(* IEC 61131-3 sources: Word/plc-course/05-boolean-logic-and-fbd/labs/starter, 3 files *)

(* ---- 05-1-pump-permissive.st ---- *)
(* Lab 05-1: Transfer pump P-101 start permissive.
   Module 05 (Boolean logic and FBD). STARTER - the declarations are done for you;
   write the logic where it says TODO, then run:
     python3 tools/plctest.py 05-boolean-logic-and-fbd/labs/starter/05-1-pump-permissive.st

   The whole lab is combinational: no seal-in, latch or timer is needed. *)

PROGRAM TransferPump
  VAR (* I/O - addresses follow the OpenPLC convention *)
    SuctionOpenLS AT %IX0.0 : BOOL;  (* Suction valve XV-100 open limit switch (ZSO-100): TRUE = fully open *)
    LSL101_NC     AT %IX0.1 : BOOL;  (* Tank low-level switch LSL-101, NC: TRUE = level above the switch (healthy) *)
    MotorFault    AT %IX0.2 : BOOL;  (* Motor protection relay fault contact, NO: TRUE = protection tripped *)
    ManualSel     AT %IX0.3 : BOOL;  (* MAN-OFF-AUTO selector, MAN contact *)
    AutoSel       AT %IX0.4 : BOOL;  (* MAN-OFF-AUTO selector, AUTO contact *)
    Demand        AT %IX0.5 : BOOL;  (* Auto demand from the process: TRUE = liquid wanted *)
    ManualRunCmd  AT %IX0.6 : BOOL;  (* Manual run command, maintained: TRUE = run *)
    Pump          AT %QX0.0 : BOOL;  (* P-101 motor starter: TRUE = run *)
    PermissiveOK  AT %QX0.1 : BOOL;  (* White "Ready" lamp: all start permissives healthy *)
    SelectorFault AT %QX0.2 : BOOL;  (* Both selector contacts made at once *)
  END_VAR
  (* You may add your own internal variables in a separate VAR block here. *)

  (* TODO: replace these placeholder lines with your logic.
     (MATIEC needs at least one statement in a program body.) *)
  PermissiveOK := FALSE;
  SelectorFault := FALSE;
  Pump := FALSE;
END_PROGRAM

CONFIGURATION Config0
  RESOURCE Res0 ON PLC
    TASK MainTask(INTERVAL := T#10ms, PRIORITY := 0);
    PROGRAM Inst0 WITH MainTask : TransferPump;
  END_RESOURCE
END_CONFIGURATION

(* ---- 05-2-two-out-of-three-vote.st ---- *)
(* Lab 05-2: Two-out-of-three (2oo3) high-pressure trip vote.
   Module 05 (Boolean logic and FBD). STARTER - the declarations are done for you;
   write the logic where it says TODO, then run:
     python3 tools/plctest.py 05-boolean-logic-and-fbd/labs/starter/05-2-two-out-of-three-vote.st

   TRAINING EXERCISE ONLY - not a design for a real safety function. *)

PROGRAM TripVote
  VAR (* I/O - addresses follow the OpenPLC convention *)
    PSHH_A_NC   AT %IX0.0 : BOOL;  (* PSHH-101A, NC: TRUE = pressure below trip setting (healthy) *)
    PSHH_B_NC   AT %IX0.1 : BOOL;  (* PSHH-101B, NC: as above *)
    PSHH_C_NC   AT %IX0.2 : BOOL;  (* PSHH-101C, NC: as above *)
    Trip        AT %QX0.0 : BOOL;  (* TRUE = at least two channels demand a trip *)
    SDVSolenoid AT %QX0.1 : BOOL;  (* SDV-100 solenoid: TRUE = energised, valve held open *)
    Discrepancy AT %QX0.2 : BOOL;  (* TRUE = the three channels do not all agree *)
    DiscA       AT %QX0.3 : BOOL;  (* TRUE = channel A disagrees with B and C *)
    DiscB       AT %QX0.4 : BOOL;  (* TRUE = channel B disagrees with A and C *)
    DiscC       AT %QX0.5 : BOOL;  (* TRUE = channel C disagrees with A and B *)
  END_VAR
  (* You may add your own internal variables in a separate VAR block here. *)

  (* TODO: replace these placeholder lines with your logic.
     (MATIEC needs at least one statement in a program body.) *)
  Trip := FALSE;
  SDVSolenoid := FALSE;
  Discrepancy := FALSE;
  DiscA := FALSE;
  DiscB := FALSE;
  DiscC := FALSE;
END_PROGRAM

CONFIGURATION Config0
  RESOURCE Res0 ON PLC
    TASK MainTask(INTERVAL := T#10ms, PRIORITY := 0);
    PROGRAM Inst0 WITH MainTask : TripVote;
  END_RESOURCE
END_CONFIGURATION

(* ---- 05-3-horn-truth-table.st ---- *)
(* Lab 05-3: From truth table to minimal logic - wet-well alarm horn.
   Module 05 (Boolean logic and FBD). STARTER - the declarations are done for you;
   write the logic where it says TODO, then run:
     python3 tools/plctest.py 05-boolean-logic-and-fbd/labs/starter/05-3-horn-truth-table.st

   Work from the truth table in the lesson (Lab 05-3). Draw the K-map on paper
   first and write your minimal expression in this comment:

     Horn = ...
*)

PROGRAM WetWellHorn
  VAR (* I/O - addresses follow the OpenPLC convention *)
    HighLevel AT %IX0.0 : BOOL;  (* High-level float relay: TRUE = level high *)
    LowLevel  AT %IX0.1 : BOOL;  (* Low-level float relay: TRUE = level low *)
    Pump1Run  AT %IX0.2 : BOOL;  (* Pump 1 running (contactor auxiliary contact) *)
    Pump2Run  AT %IX0.3 : BOOL;  (* Pump 2 running (contactor auxiliary contact) *)
    Horn      AT %QX0.0 : BOOL;  (* Wet-well alarm horn *)
  END_VAR

  (* TODO: replace this placeholder line with your minimal logic.
     (MATIEC needs at least one statement in a program body.) *)
  Horn := FALSE;
END_PROGRAM

CONFIGURATION Config0
  RESOURCE Res0 ON PLC
    TASK MainTask(INTERVAL := T#10ms, PRIORITY := 0);
    PROGRAM Inst0 WITH MainTask : WetWellHorn;
  END_RESOURCE
END_CONFIGURATION
